FUNCTION_BLOCK Manueller_Betrieb
VAR_INPUT
	Kein_Notaus : BOOL;
	//Taster auf Bedienfeld
	Hydraulik_EIN : BOOL;
	Hydraulik_AUS : BOOL;
	Kettenschmierung_Manuell_EIN : BOOL;
	Zufuehrer_Vor : BOOL;
	Zufuehrer_Rueck : BOOL;
	Stammklemmer_Oben_Hoch : BOOL;
	Stammklemmer_Oben_Runter : BOOL;
	Stammklemmer_Unten_Hoch : BOOL;
	Stammklemmer_Unten_Runter : BOOL;
	Saege_EIN : BOOL;
	Saege_AUS : BOOL;
	Saege_Hoch : BOOL;
	Saege_Runter : BOOL;
	
	
	//Eingänge Sensorik
	//Zuführer
	Endl_Zufuehrer_Hinten : BOOL;
	Endl_Zufuehrer_Vorne : BOOL;
	Vorposition_Zufuehrer : BOOL;
	//Stammklemmung Oben
	Endl_Obere_Stammklemmung_Oben : BOOL;
	Endl_Obere_Stammklemmung_Unten : BOOL;
	Endl_Tastschiene : BOOL;
	Schaltausg_Druckschalter_Obere_Klemmung : BOOL;
	//Stammklemmung Unten
	Endl_Untere_Stammklemmung_Oben : BOOL;
	Endl_Untere_Stammklemmung_Unten : BOOL;
	//Säge
	Endl_Saege_Oben : BOOL;
	Endl_Saege_Unten : BOOL;
END_VAR
VAR_OUTPUT
	//Ausgänge Hydraulik
	QStammklemmung_Oben_Hoch : BOOL;
	QStammklemmung_Oben_Runter : BOOL;
	QStammklemmung_Unten_Hoch : BOOL;
	QStammklemmung_Unten_Runter : BOOL;
	QSaege_Senken : BOOL;
	QSaege_Heben : BOOL;
	//Ausgänge Schalten
	QHydraulikpumpe_EIN : BOOL;
	QZufuehrer_Antrieb_vor : BOOL;
	QZufuehrer_Antrieb_Rueck : BOOL;
	QSaege_Antrieb_Ein : BOOL;
	QKettenschmierung_EIN : BOOL;
	//Ausgänge Daten
	//FU DATEN
END_VAR
VAR_IN_OUT
	
	
END_VAR
VAR
END_VAR

QStammklemmung_Oben_Hoch :=
QStammklemmung_Oben_Runter := 
QStammklemmung_Unten_Hoch := 
QStammklemmung_Unten_Runter := 
QSaege_Senken := 
QSaege_Heben := 
QZufuehrer_Antrieb_vor := 
QZufuehrer_Antrieb_Rueck := 
QSaege_Antrieb_Ein := 
QKettenschmierung_EIN := FALSE;

IF Hydraulik_EIN THEN
	QHydraulikpumpe_EIN := TRUE;
END_IF

IF Hydraulik_AUS THEN
	QHydraulikpumpe_EIN := FALSE;
END_IF

//Funktionen mit Hydraulik
IF QHydraulikpumpe_EIN THEN
	QStammklemmung_Oben_Hoch := Stammklemmer_Oben_Hoch AND NOT Stammklemmer_Oben_Runter;
	QStammklemmung_Oben_Runter := Stammklemmer_Oben_Runter AND NOT Stammklemmer_Oben_Hoch;
	QStammklemmung_Unten_Hoch := Stammklemmer_Unten_Hoch AND NOT Stammklemmer_Unten_Runter;
	QStammklemmung_Unten_Runter := Stammklemmer_Unten_Runter AND NOT Stammklemmer_Unten_Hoch;
	QSaege_Senken := Saege_Runter AND NOT Saege_Hoch AND NOT Saege_Hoch;
	QSaege_Heben := Saege_Hoch AND NOT Saege_Runter AND NOT Saege_Runter;
END_IF

//Funktionen ohne Hydraulik
IF Hydraulik_EIN THEN
	QHydraulikpumpe_EIN := TRUE;
ELSIF Hydraulik_AUS THEN
	QHydraulikpumpe_EIN := FALSE;
END_IF

QZufuehrer_Antrieb_vor := Zufuehrer_Vor AND NOT Zufuehrer_Rueck;
QZufuehrer_Antrieb_Rueck := Zufuehrer_Rueck AND NOT Zufuehrer_Vor;

QSaege_Antrieb_Ein := Saege_EIN;

END_FUNCTION_BLOCK

(* stored: Version 1.1.0.1, ProductVersion 3.1.4024.16
   POU Manueller_Betrieb: Id {ac3c5180-7042-481e-a944-4bd75763f607}, SpecialFunc None *)
